PROGRAM MAIN
VAR
END_VAR

END_PROGRAM

(* stored: Version 1.1.0.1
   POU MAIN: Id {b398755d-16bf-45e3-b3a1-406c203abc04} *)
